// TIA Portal V18 export
FUNCTION "AHUEqpCtrl" : Void   // FC60301, LAD
{ S7_Optimized_Access := 'TRUE' }
VERSION : 0.1
// Type                                             Control State
// 0 = no ctrl                                             0 = Stopped/Closed/NA
// 1 = Proxi/Adaptation                           1 = 100%/FullyOpened/ 
// 2=                                                           2 = RegulationEnable
// stored: AutoNumber false, IsIECCheckEnabled false, SetENOAutomatically false, UDAEnableTagReadback false
   VAR_INPUT
      iUnitID : Int;
      cActualUnitState : Byte;
      cActualSeason : Byte;
      cFanType : Byte;
      cExtractDumperType : Byte;
      cMixingDumperType : Byte;
      cHeaterType : Byte;
      cCoolerType : Byte;
      cWHUType : Byte;
   END_VAR
   VAR_OUTPUT
      cFanCtrlState : Byte;
      cExtractCtrlState : Byte;
      cMixingCtrlState : Byte;
      cHeaterCtrlState : Byte;
      cCoolerCtrlState : Byte;
      cWHUCtrlState : Byte;
   END_VAR
BEGIN

REGION Network 1 (SCL): Fan
   CASE #cFanType OF
       0:  //disable
           #cFanCtrlState := 0;
       ELSE  // Active
           #cFanCtrlState := 2;
   END_CASE;
END_REGION

REGION Network 2 (SCL): Extract Dumper
   CASE #cExtractDumperType OF
       0:  //disable
           #cExtractCtrlState := 0;
       ELSE  // Active
           CASE #cActualSeason OF
               0:  // Winter
                   #cExtractCtrlState := 0;//Blocked
               1:  // Summer
                   #cExtractCtrlState := 0;//Auto
               ELSE  //Midseason
                   #cExtractCtrlState := 2;//Auto
           END_CASE;
   END_CASE;
END_REGION

REGION Network 3 (SCL): Mixing Dumper
   CASE #cMixingDumperType OF
       0:  //disable
           #cMixingCtrlState := 0;
       ELSE  // Active
           IF #cActualUnitState = 4 THEN // 100% recycling mode
               #cMixingCtrlState := 1;
           ELSE
               #cMixingCtrlState := 2;
           END_IF;
   END_CASE;
END_REGION

REGION Network 4 (SCL): Heater
   CASE #cHeaterType OF
       0:  //disable
           #cHeaterCtrlState := 0;
       ELSE  // Active
           IF #cActualUnitState =2  THEN //Preheating
               #cHeaterCtrlState := 1;
           ELSE

               CASE #cActualSeason OF
                   0:  // Winter
                       #cHeaterCtrlState := 2;//Auto
                   1:  // Summer
                       #cHeaterCtrlState := 0;//Blocked
                   ELSE  //Midseason
                       #cHeaterCtrlState := 2;//Auto
               END_CASE;
           END_IF;
   END_CASE;
END_REGION

REGION Network 5 (SCL): Cooler
   CASE #cCoolerType OF
       0:  //disable
           #cCoolerCtrlState := 0;
       ELSE  // Active
           CASE #cActualSeason OF
               0:  //Winter
                   #cCoolerCtrlState := 0;//Blocked
               1:  // Summer
                   #cCoolerCtrlState := 2;//Auto
               ELSE  //Midseason
                   #cCoolerCtrlState := 2;//Auto
           END_CASE;
   END_CASE;
END_REGION

REGION Network 6 (SCL): WHU
   CASE #cWHUType OF
       0:  //disable
           #cWHUCtrlState := 0;
       ELSE  // Active
           CASE #cActualSeason OF
               0:  // Winter
                   #cWHUCtrlState := 2;//Auto
               1:  // Summer
                   #cWHUCtrlState := 0;//Blocked
               ELSE  //Midseason
                   #cWHUCtrlState := 2;//Auto
           END_CASE;
   END_CASE;
END_REGION
END_FUNCTION
